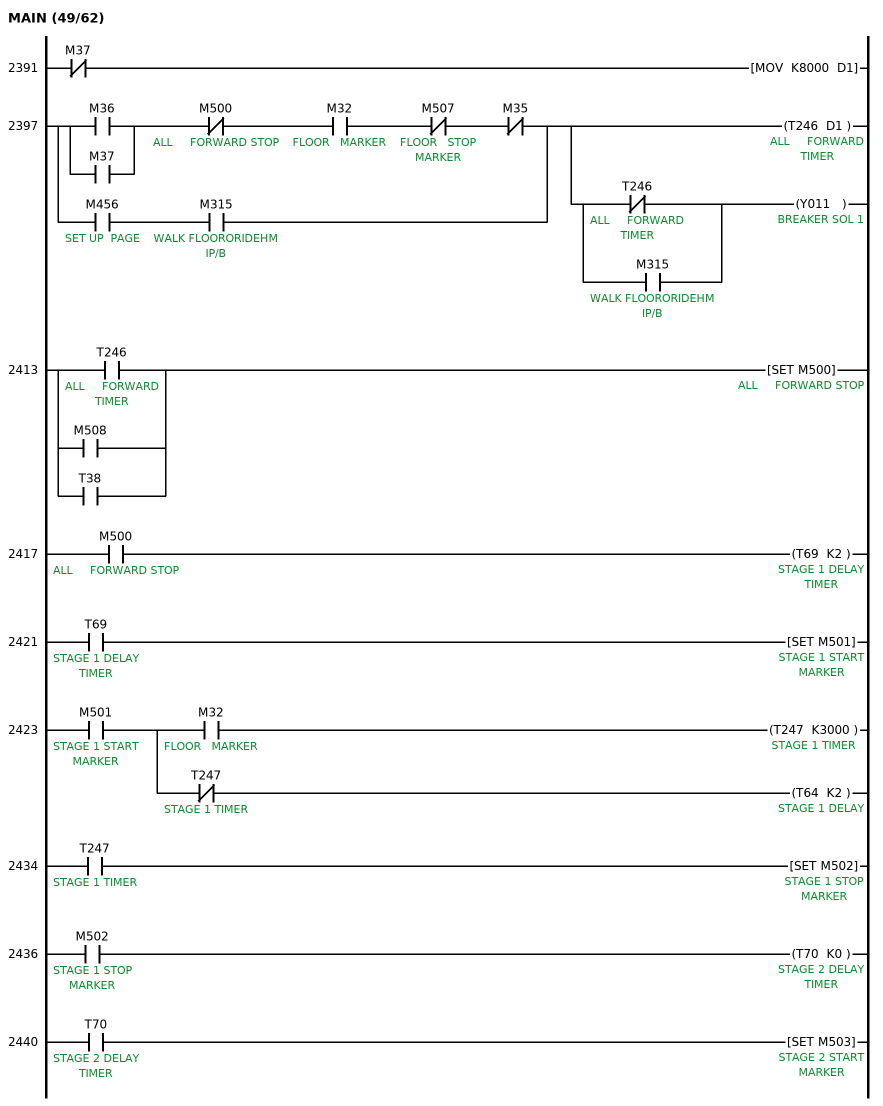
2391  LDI     M37
      MOV     K8000 D1
2397  LD      M36
      OR      M37
      ANI     M500  ; ALL     FORWARD STOP
      AND     M32  ; FLOOR   MARKER
      ANI     M507  ; FLOOR   STOP    MARKER
      ANI     M35
      LD      M456  ; SET UP  PAGE
      AND     M315  ; WALK FLOORORIDEHMIP/B
      ORB
      OUT     T246 D1  ; ALL     FORWARD TIMER
      LDI     T246  ; ALL     FORWARD TIMER
      OR      M315  ; WALK FLOORORIDEHMIP/B
      ANB
      OUT     Y011  ; BREAKER SOL 1
2413  LD      T246  ; ALL     FORWARD TIMER
      OR      M508
      OR      T38
      SET     M500  ; ALL     FORWARD STOP
2417  LD      M500  ; ALL     FORWARD STOP
      OUT     T69 K2  ; STAGE 1 DELAY   TIMER
2421  LD      T69  ; STAGE 1 DELAY   TIMER
      SET     M501  ; STAGE 1 START   MARKER
2423  LD      M501  ; STAGE 1 START   MARKER
      MPS
      AND     M32  ; FLOOR   MARKER
      OUT     T247 K3000  ; STAGE 1 TIMER
      MPP
      ANI     T247  ; STAGE 1 TIMER
      OUT     T64 K2  ; STAGE 1 DELAY
2434  LD      T247  ; STAGE 1 TIMER
      SET     M502  ; STAGE 1 STOP    MARKER
2436  LD      M502  ; STAGE 1 STOP    MARKER
      OUT     T70 K0  ; STAGE 2 DELAY   TIMER
2440  LD      T70  ; STAGE 2 DELAY   TIMER
      SET     M503  ; STAGE 2 START   MARKER
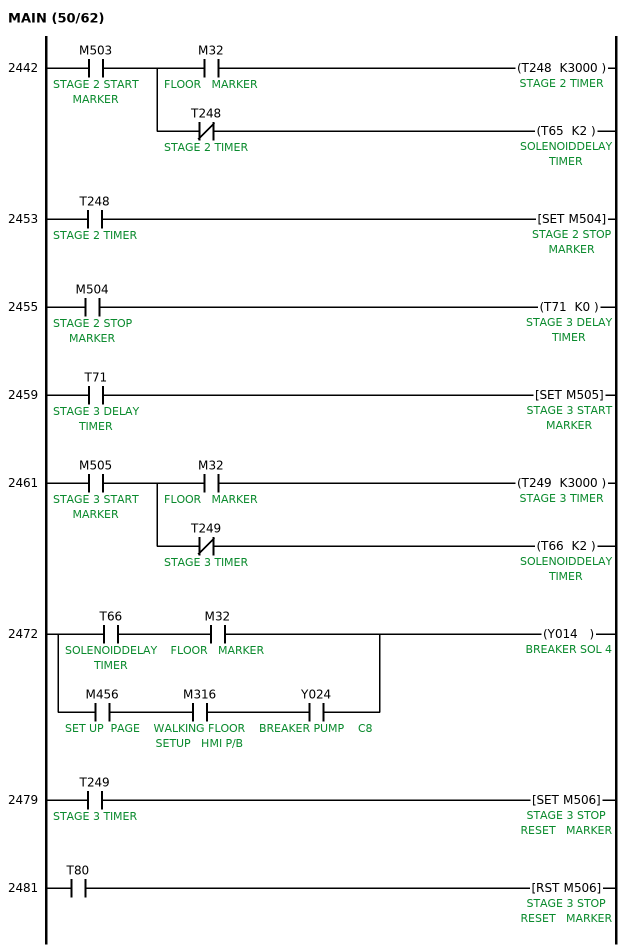
2442  LD      M503  ; STAGE 2 START   MARKER
      MPS
      AND     M32  ; FLOOR   MARKER
      OUT     T248 K3000  ; STAGE 2 TIMER
      MPP
      ANI     T248  ; STAGE 2 TIMER
      OUT     T65 K2  ; SOLENOIDDELAY   TIMER
2453  LD      T248  ; STAGE 2 TIMER
      SET     M504  ; STAGE 2 STOP    MARKER
2455  LD      M504  ; STAGE 2 STOP    MARKER
      OUT     T71 K0  ; STAGE 3 DELAY   TIMER
2459  LD      T71  ; STAGE 3 DELAY   TIMER
      SET     M505  ; STAGE 3 START   MARKER
2461  LD      M505  ; STAGE 3 START   MARKER
      MPS
      AND     M32  ; FLOOR   MARKER
      OUT     T249 K3000  ; STAGE 3 TIMER
      MPP
      ANI     T249  ; STAGE 3 TIMER
      OUT     T66 K2  ; SOLENOIDDELAY   TIMER
2472  LD      T66  ; SOLENOIDDELAY   TIMER
      AND     M32  ; FLOOR   MARKER
      LD      M456  ; SET UP  PAGE
      AND     M316  ; WALKING FLOOR   SETUP   HMI P/B
      AND     Y024  ; BREAKER PUMP    C8
      ORB
      OUT     Y014  ; BREAKER SOL 4
2479  LD      T249  ; STAGE 3 TIMER
      SET     M506  ; STAGE 3 STOP    RESET   MARKER
2481  LD      T80
      RST     M506  ; STAGE 3 STOP    RESET   MARKER
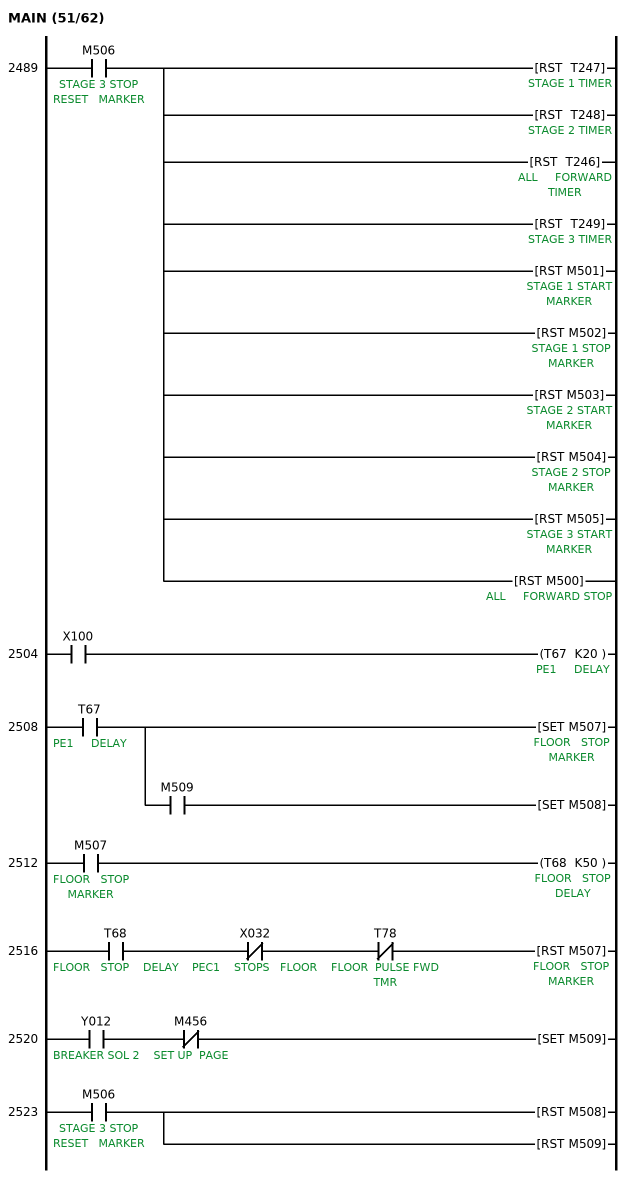
2489  LD      M506  ; STAGE 3 STOP    RESET   MARKER
      RST     T247  ; STAGE 1 TIMER
      RST     T248  ; STAGE 2 TIMER
      RST     T246  ; ALL     FORWARD TIMER
      RST     T249  ; STAGE 3 TIMER
      RST     M501  ; STAGE 1 START   MARKER
      RST     M502  ; STAGE 1 STOP    MARKER
      RST     M503  ; STAGE 2 START   MARKER
      RST     M504  ; STAGE 2 STOP    MARKER
      RST     M505  ; STAGE 3 START   MARKER
      RST     M500  ; ALL     FORWARD STOP
2504  LD      X100
      OUT     T67 K20  ; PE1     DELAY
2508  LD      T67  ; PE1     DELAY
      SET     M507  ; FLOOR   STOP    MARKER
      AND     M509
      SET     M508
2512  LD      M507  ; FLOOR   STOP    MARKER
      OUT     T68 K50  ; FLOOR   STOP    DELAY
2516  LD      T68  ; FLOOR   STOP    DELAY
      ANI     X032  ; PEC1    STOPS   FLOOR
      ANI     T78  ; FLOOR  PULSE FWD TMR
      RST     M507  ; FLOOR   STOP    MARKER
2520  LD      Y012  ; BREAKER SOL 2
      ANI     M456  ; SET UP  PAGE
      SET     M509
2523  LD      M506  ; STAGE 3 STOP    RESET   MARKER
      RST     M508
      RST     M509
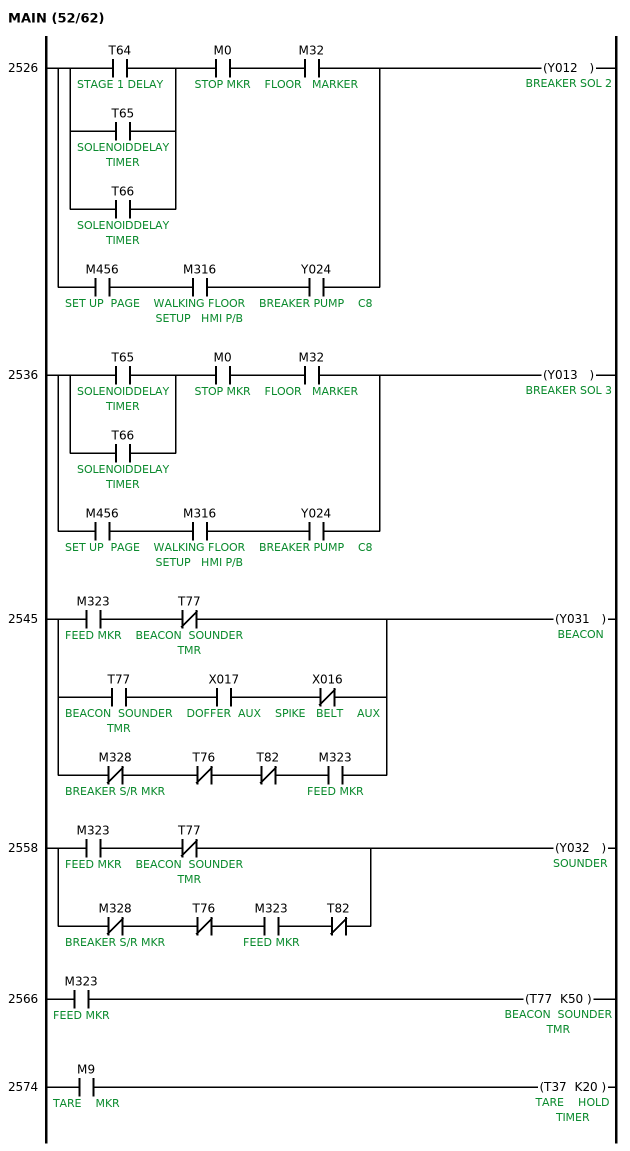
2526  LD      T64  ; STAGE 1 DELAY
      OR      T65  ; SOLENOIDDELAY   TIMER
      OR      T66  ; SOLENOIDDELAY   TIMER
      AND     M0  ; STOP MKR
      AND     M32  ; FLOOR   MARKER
      LD      M456  ; SET UP  PAGE
      AND     M316  ; WALKING FLOOR   SETUP   HMI P/B
      AND     Y024  ; BREAKER PUMP    C8
      ORB
      OUT     Y012  ; BREAKER SOL 2
2536  LD      T65  ; SOLENOIDDELAY   TIMER
      OR      T66  ; SOLENOIDDELAY   TIMER
      AND     M0  ; STOP MKR
      AND     M32  ; FLOOR   MARKER
      LD      M456  ; SET UP  PAGE
      AND     M316  ; WALKING FLOOR   SETUP   HMI P/B
      AND     Y024  ; BREAKER PUMP    C8
      ORB
      OUT     Y013  ; BREAKER SOL 3
2545  LD      M323  ; FEED MKR
      ANI     T77  ; BEACON  SOUNDER TMR
      LD      T77  ; BEACON  SOUNDER TMR
      AND     X017  ; DOFFER  AUX
      ANI     X016  ; SPIKE   BELT    AUX
      ORB
      LDI     M328  ; BREAKER S/R MKR
      ANI     T76
      ANI     T82
      AND     M323  ; FEED MKR
      ORB
      OUT     Y031  ; BEACON
2558  LD      M323  ; FEED MKR
      ANI     T77  ; BEACON  SOUNDER TMR
      LDI     M328  ; BREAKER S/R MKR
      ANI     T76
      AND     M323  ; FEED MKR
      ANI     T82
      ORB
      OUT     Y032  ; SOUNDER
2566  LD      M323  ; FEED MKR
      OUT     T77 K50  ; BEACON  SOUNDER TMR
2574  LD      M9  ; TARE    MKR
      OUT     T37 K20  ; TARE    HOLD    TIMER
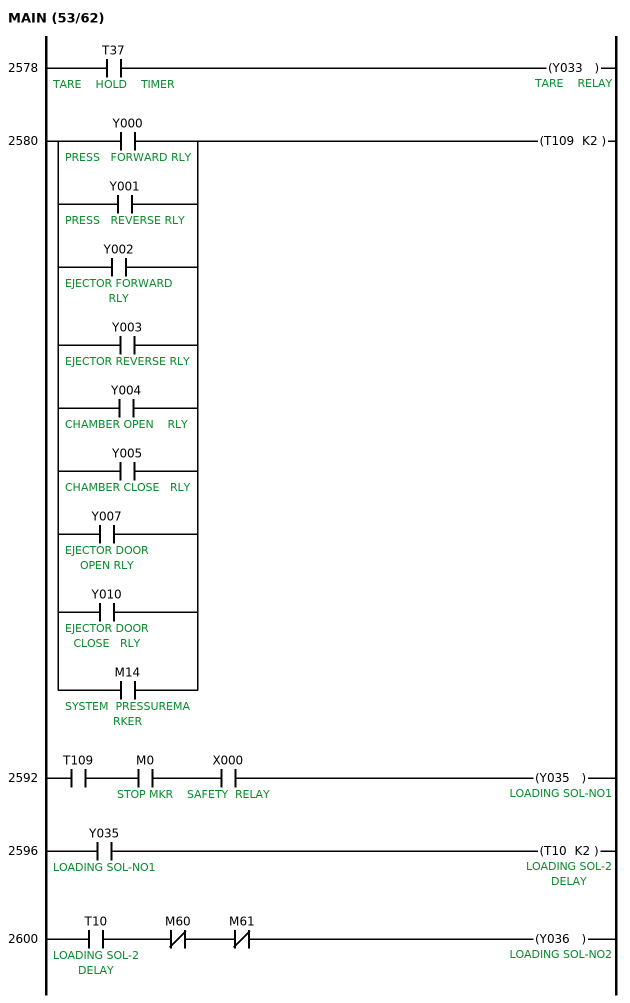
2578  LD      T37  ; TARE    HOLD    TIMER
      OUT     Y033  ; TARE    RELAY
2580  LD      Y000  ; PRESS   FORWARD RLY
      OR      Y001  ; PRESS   REVERSE RLY
      OR      Y002  ; EJECTOR FORWARD RLY
      OR      Y003  ; EJECTOR REVERSE RLY
      OR      Y004  ; CHAMBER OPEN    RLY
      OR      Y005  ; CHAMBER CLOSE   RLY
      OR      Y007  ; EJECTOR DOOR    OPEN RLY
      OR      Y010  ; EJECTOR DOOR    CLOSE   RLY
      OR      M14  ; SYSTEM  PRESSUREMARKER
      OUT     T109 K2
2592  LD      T109
      AND     M0  ; STOP MKR
      AND     X000  ; SAFETY  RELAY
      OUT     Y035  ; LOADING SOL-NO1
2596  LD      Y035  ; LOADING SOL-NO1
      OUT     T10 K2  ; LOADING SOL-2   DELAY
2600  LD      T10  ; LOADING SOL-2   DELAY
      ANI     M60
      ANI     M61
      OUT     Y036  ; LOADING SOL-NO2
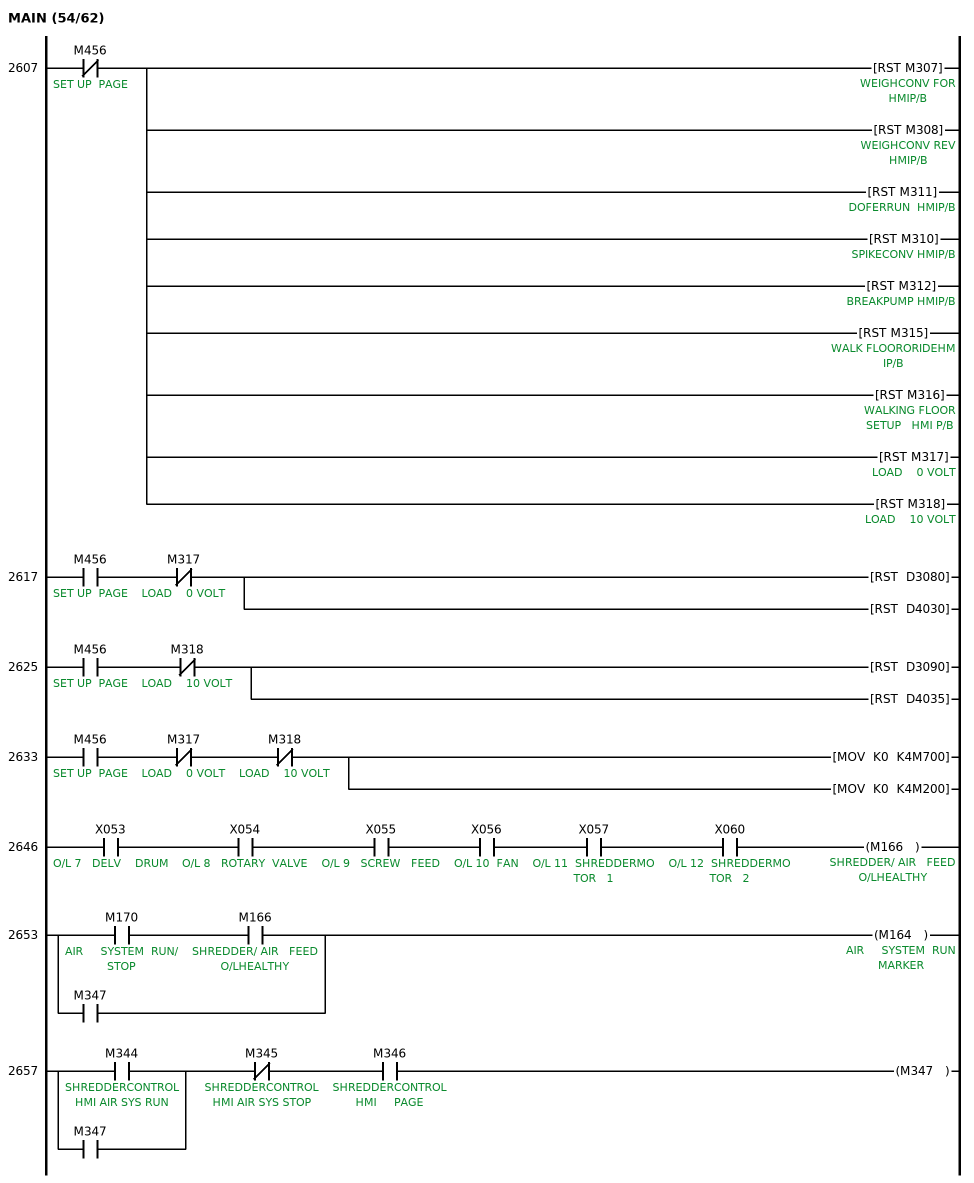
2607  LDI     M456  ; SET UP  PAGE
      RST     M307  ; WEIGHCONV FOR   HMIP/B
      RST     M308  ; WEIGHCONV REV   HMIP/B
      RST     M311  ; DOFERRUN  HMIP/B
      RST     M310  ; SPIKECONV HMIP/B
      RST     M312  ; BREAKPUMP HMIP/B
      RST     M315  ; WALK FLOORORIDEHMIP/B
      RST     M316  ; WALKING FLOOR   SETUP   HMI P/B
      RST     M317  ; LOAD    0 VOLT
      RST     M318  ; LOAD    10 VOLT
2617  LD      M456  ; SET UP  PAGE
      ANI     M317  ; LOAD    0 VOLT
      RST     D3080
      RST     D4030
2625  LD      M456  ; SET UP  PAGE
      ANI     M318  ; LOAD    10 VOLT
      RST     D3090
      RST     D4035
2633  LD      M456  ; SET UP  PAGE
      ANI     M317  ; LOAD    0 VOLT
      ANI     M318  ; LOAD    10 VOLT
      MOV     K0 K4M700
      MOV     K0 K4M200
2646  LD      X053  ; O/L 7   DELV    DRUM
      AND     X054  ; O/L 8   ROTARY  VALVE
      AND     X055  ; O/L 9   SCREW   FEED
      AND     X056  ; O/L 10  FAN
      AND     X057  ; O/L 11  SHREDDERMOTOR   1
      AND     X060  ; O/L 12  SHREDDERMOTOR   2
      OUT     M166  ; SHREDDER/ AIR   FEED O/LHEALTHY
2653  LD      M170  ; AIR     SYSTEM  RUN/    STOP
      AND     M166  ; SHREDDER/ AIR   FEED O/LHEALTHY
      OR      M347
      OUT     M164  ; AIR     SYSTEM  RUN     MARKER
2657  LD      M344  ; SHREDDERCONTROL HMI AIR SYS RUN
      OR      M347
      ANI     M345  ; SHREDDERCONTROL HMI AIR SYS STOP
      AND     M346  ; SHREDDERCONTROL HMI     PAGE
      OUT     M347
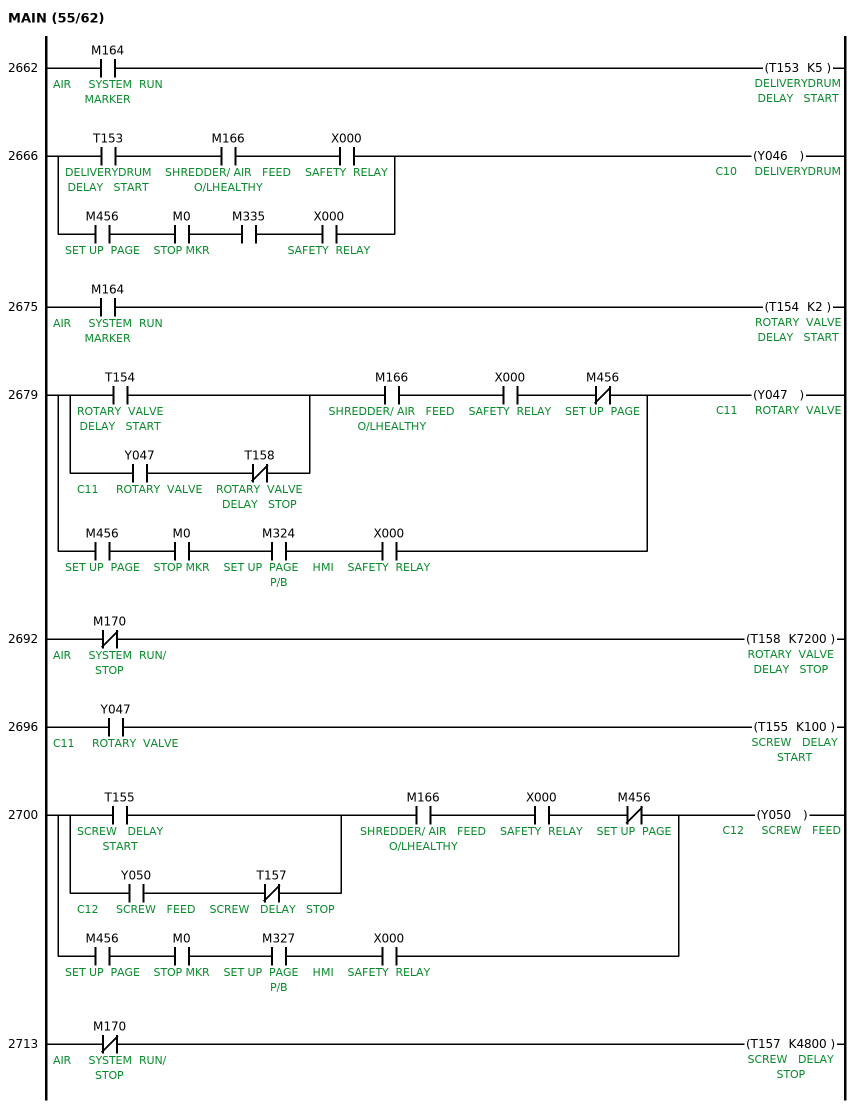
2662  LD      M164  ; AIR     SYSTEM  RUN     MARKER
      OUT     T153 K5  ; DELIVERYDRUM    DELAY   START
2666  LD      T153  ; DELIVERYDRUM    DELAY   START
      AND     M166  ; SHREDDER/ AIR   FEED O/LHEALTHY
      AND     X000  ; SAFETY  RELAY
      LD      M456  ; SET UP  PAGE
      AND     M0  ; STOP MKR
      AND     M335
      AND     X000  ; SAFETY  RELAY
      ORB
      OUT     Y046  ; C10     DELIVERYDRUM
2675  LD      M164  ; AIR     SYSTEM  RUN     MARKER
      OUT     T154 K2  ; ROTARY  VALVE   DELAY   START
2679  LD      T154  ; ROTARY  VALVE   DELAY   START
      LD      Y047  ; C11     ROTARY  VALVE
      ANI     T158  ; ROTARY  VALVE   DELAY   STOP
      ORB
      AND     M166  ; SHREDDER/ AIR   FEED O/LHEALTHY
      AND     X000  ; SAFETY  RELAY
      ANI     M456  ; SET UP  PAGE
      LD      M456  ; SET UP  PAGE
      AND     M0  ; STOP MKR
      AND     M324  ; SET UP  PAGE    HMI P/B
      AND     X000  ; SAFETY  RELAY
      ORB
      OUT     Y047  ; C11     ROTARY  VALVE
2692  LDI     M170  ; AIR     SYSTEM  RUN/    STOP
      OUT     T158 K7200  ; ROTARY  VALVE   DELAY   STOP
2696  LD      Y047  ; C11     ROTARY  VALVE
      OUT     T155 K100  ; SCREW   DELAY   START
2700  LD      T155  ; SCREW   DELAY   START
      LD      Y050  ; C12     SCREW   FEED
      ANI     T157  ; SCREW   DELAY   STOP
      ORB
      AND     M166  ; SHREDDER/ AIR   FEED O/LHEALTHY
      AND     X000  ; SAFETY  RELAY
      ANI     M456  ; SET UP  PAGE
      LD      M456  ; SET UP  PAGE
      AND     M0  ; STOP MKR
      AND     M327  ; SET UP  PAGE    HMI P/B
      AND     X000  ; SAFETY  RELAY
      ORB
      OUT     Y050  ; C12     SCREW   FEED
2713  LDI     M170  ; AIR     SYSTEM  RUN/    STOP
      OUT     T157 K4800  ; SCREW   DELAY   STOP
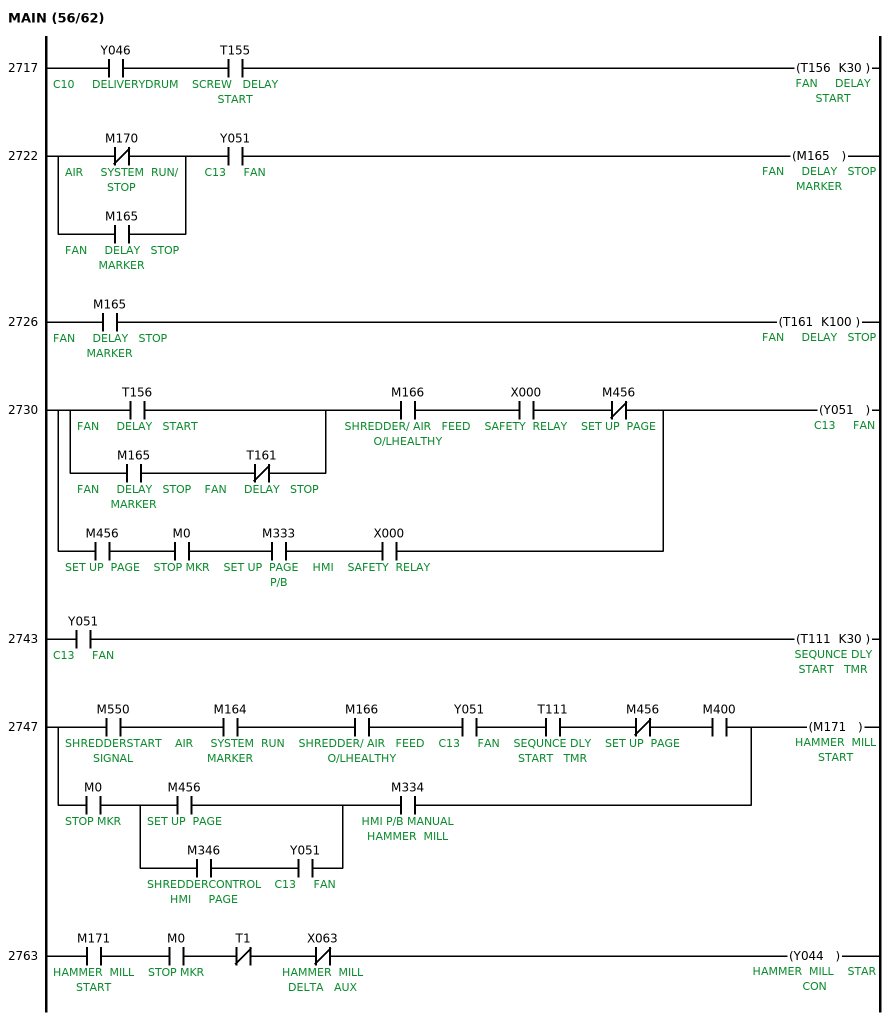
2717  LD      Y046  ; C10     DELIVERYDRUM
      AND     T155  ; SCREW   DELAY   START
      OUT     T156 K30  ; FAN     DELAY   START
2722  LDI     M170  ; AIR     SYSTEM  RUN/    STOP
      OR      M165  ; FAN     DELAY   STOP    MARKER
      AND     Y051  ; C13     FAN
      OUT     M165  ; FAN     DELAY   STOP    MARKER
2726  LD      M165  ; FAN     DELAY   STOP    MARKER
      OUT     T161 K100  ; FAN     DELAY   STOP
2730  LD      T156  ; FAN     DELAY   START
      LD      M165  ; FAN     DELAY   STOP    MARKER
      ANI     T161  ; FAN     DELAY   STOP
      ORB
      AND     M166  ; SHREDDER/ AIR   FEED O/LHEALTHY
      AND     X000  ; SAFETY  RELAY
      ANI     M456  ; SET UP  PAGE
      LD      M456  ; SET UP  PAGE
      AND     M0  ; STOP MKR
      AND     M333  ; SET UP  PAGE    HMI P/B
      AND     X000  ; SAFETY  RELAY
      ORB
      OUT     Y051  ; C13     FAN
2743  LD      Y051  ; C13     FAN
      OUT     T111 K30  ; SEQUNCE DLY     START   TMR
2747  LD      M550  ; SHREDDERSTART   SIGNAL
      AND     M164  ; AIR     SYSTEM  RUN     MARKER
      AND     M166  ; SHREDDER/ AIR   FEED O/LHEALTHY
      AND     Y051  ; C13     FAN
      AND     T111  ; SEQUNCE DLY     START   TMR
      ANI     M456  ; SET UP  PAGE
      AND     M400
      LD      M0  ; STOP MKR
      LD      M456  ; SET UP  PAGE
      LD      M346  ; SHREDDERCONTROL HMI     PAGE
      AND     Y051  ; C13     FAN
      ORB
      ANB
      AND     M334  ; HMI P/B MANUAL  HAMMER  MILL
      ORB
      OUT     M171  ; HAMMER  MILL    START
2763  LD      M171  ; HAMMER  MILL    START
      AND     M0  ; STOP MKR
      ANI     T1
      ANI     X063  ; HAMMER  MILL    DELTA   AUX
      OUT     Y044  ; HAMMER  MILL    STAR    CON
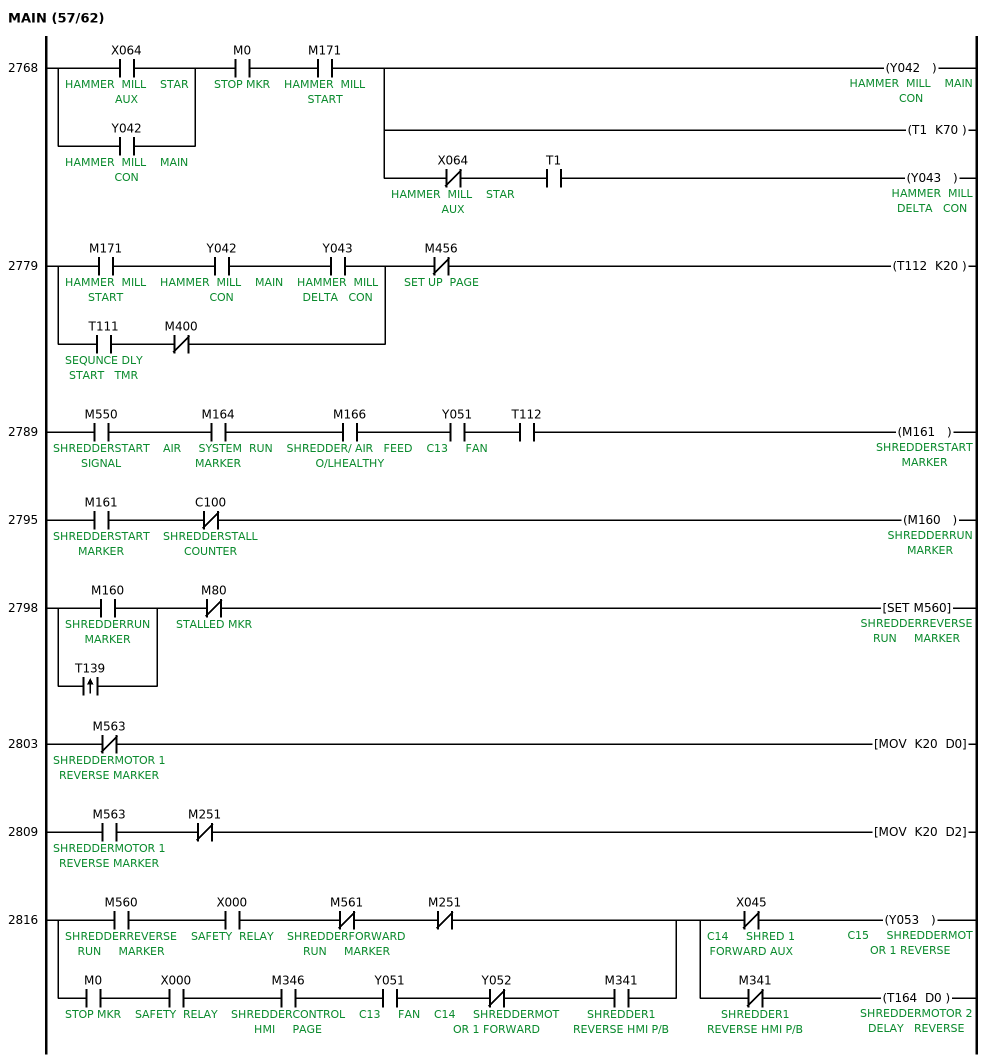
2768  LD      X064  ; HAMMER  MILL    STAR    AUX
      OR      Y042  ; HAMMER  MILL    MAIN    CON
      AND     M0  ; STOP MKR
      AND     M171  ; HAMMER  MILL    START
      OUT     Y042  ; HAMMER  MILL    MAIN    CON
      OUT     T1 K70
      ANI     X064  ; HAMMER  MILL    STAR    AUX
      AND     T1
      OUT     Y043  ; HAMMER  MILL    DELTA   CON
2779  LD      M171  ; HAMMER  MILL    START
      AND     Y042  ; HAMMER  MILL    MAIN    CON
      AND     Y043  ; HAMMER  MILL    DELTA   CON
      LD      T111  ; SEQUNCE DLY     START   TMR
      ANI     M400
      ORB
      ANI     M456  ; SET UP  PAGE
      OUT     T112 K20
2789  LD      M550  ; SHREDDERSTART   SIGNAL
      AND     M164  ; AIR     SYSTEM  RUN     MARKER
      AND     M166  ; SHREDDER/ AIR   FEED O/LHEALTHY
      AND     Y051  ; C13     FAN
      AND     T112
      OUT     M161  ; SHREDDERSTART   MARKER
2795  LD      M161  ; SHREDDERSTART   MARKER
      ANI     C100  ; SHREDDERSTALL   COUNTER
      OUT     M160  ; SHREDDERRUN     MARKER
2798  LD      M160  ; SHREDDERRUN     MARKER
      ORP     T139
      ANI     M80  ; STALLED MKR
      SET     M560  ; SHREDDERREVERSE RUN     MARKER
2803  LDI     M563  ; SHREDDERMOTOR 1 REVERSE MARKER
      MOV     K20 D0
2809  LD      M563  ; SHREDDERMOTOR 1 REVERSE MARKER
      ANI     M251
      MOV     K20 D2
2816  LD      M560  ; SHREDDERREVERSE RUN     MARKER
      AND     X000  ; SAFETY  RELAY
      ANI     M561  ; SHREDDERFORWARD RUN     MARKER
      ANI     M251
      LD      M0  ; STOP MKR
      AND     X000  ; SAFETY  RELAY
      AND     M346  ; SHREDDERCONTROL HMI     PAGE
      AND     Y051  ; C13     FAN
      ANI     Y052  ; C14     SHREDDERMOTOR 1 FORWARD
      AND     M341  ; SHREDDER1       REVERSE HMI P/B
      ORB
      MPS
      ANI     X045  ; C14     SHRED 1 FORWARD AUX
      OUT     Y053  ; C15     SHREDDERMOTOR 1 REVERSE
      MPP
      ANI     M341  ; SHREDDER1       REVERSE HMI P/B
      OUT     T164 D0  ; SHREDDERMOTOR 2 DELAY   REVERSE
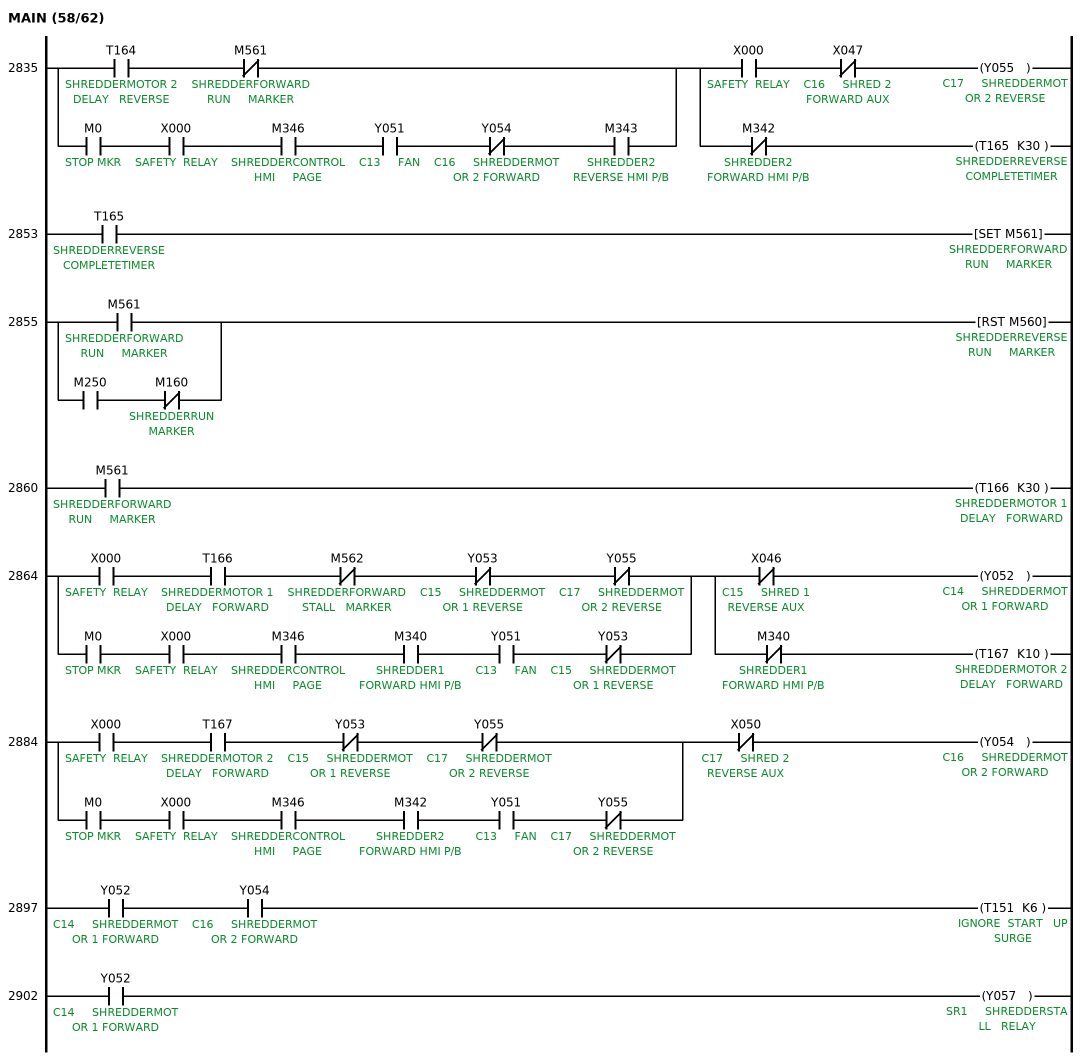
2835  LD      T164  ; SHREDDERMOTOR 2 DELAY   REVERSE
      ANI     M561  ; SHREDDERFORWARD RUN     MARKER
      LD      M0  ; STOP MKR
      AND     X000  ; SAFETY  RELAY
      AND     M346  ; SHREDDERCONTROL HMI     PAGE
      AND     Y051  ; C13     FAN
      ANI     Y054  ; C16     SHREDDERMOTOR 2 FORWARD
      AND     M343  ; SHREDDER2       REVERSE HMI P/B
      ORB
      MPS
      AND     X000  ; SAFETY  RELAY
      ANI     X047  ; C16     SHRED 2 FORWARD AUX
      OUT     Y055  ; C17     SHREDDERMOTOR 2 REVERSE
      MPP
      ANI     M342  ; SHREDDER2       FORWARD HMI P/B
      OUT     T165 K30  ; SHREDDERREVERSE COMPLETETIMER
2853  LD      T165  ; SHREDDERREVERSE COMPLETETIMER
      SET     M561  ; SHREDDERFORWARD RUN     MARKER
2855  LD      M561  ; SHREDDERFORWARD RUN     MARKER
      LD      M250
      ANI     M160  ; SHREDDERRUN     MARKER
      ORB
      RST     M560  ; SHREDDERREVERSE RUN     MARKER
2860  LD      M561  ; SHREDDERFORWARD RUN     MARKER
      OUT     T166 K30  ; SHREDDERMOTOR 1 DELAY   FORWARD
2864  LD      X000  ; SAFETY  RELAY
      AND     T166  ; SHREDDERMOTOR 1 DELAY   FORWARD
      ANI     M562  ; SHREDDERFORWARD STALL   MARKER
      ANI     Y053  ; C15     SHREDDERMOTOR 1 REVERSE
      ANI     Y055  ; C17     SHREDDERMOTOR 2 REVERSE
      LD      M0  ; STOP MKR
      AND     X000  ; SAFETY  RELAY
      AND     M346  ; SHREDDERCONTROL HMI     PAGE
      AND     M340  ; SHREDDER1       FORWARD HMI P/B
      AND     Y051  ; C13     FAN
      ANI     Y053  ; C15     SHREDDERMOTOR 1 REVERSE
      ORB
      MPS
      ANI     X046  ; C15     SHRED 1 REVERSE AUX
      OUT     Y052  ; C14     SHREDDERMOTOR 1 FORWARD
      MPP
      ANI     M340  ; SHREDDER1       FORWARD HMI P/B
      OUT     T167 K10  ; SHREDDERMOTOR 2 DELAY   FORWARD
2884  LD      X000  ; SAFETY  RELAY
      AND     T167  ; SHREDDERMOTOR 2 DELAY   FORWARD
      ANI     Y053  ; C15     SHREDDERMOTOR 1 REVERSE
      ANI     Y055  ; C17     SHREDDERMOTOR 2 REVERSE
      LD      M0  ; STOP MKR
      AND     X000  ; SAFETY  RELAY
      AND     M346  ; SHREDDERCONTROL HMI     PAGE
      AND     M342  ; SHREDDER2       FORWARD HMI P/B
      AND     Y051  ; C13     FAN
      ANI     Y055  ; C17     SHREDDERMOTOR 2 REVERSE
      ORB
      ANI     X050  ; C17     SHRED 2 REVERSE AUX
      OUT     Y054  ; C16     SHREDDERMOTOR 2 FORWARD
2897  LD      Y052  ; C14     SHREDDERMOTOR 1 FORWARD
      AND     Y054  ; C16     SHREDDERMOTOR 2 FORWARD
      OUT     T151 K6  ; IGNORE  START   UP      SURGE
2902  LD      Y052  ; C14     SHREDDERMOTOR 1 FORWARD
      OUT     Y057  ; SR1     SHREDDERSTALL   RELAY
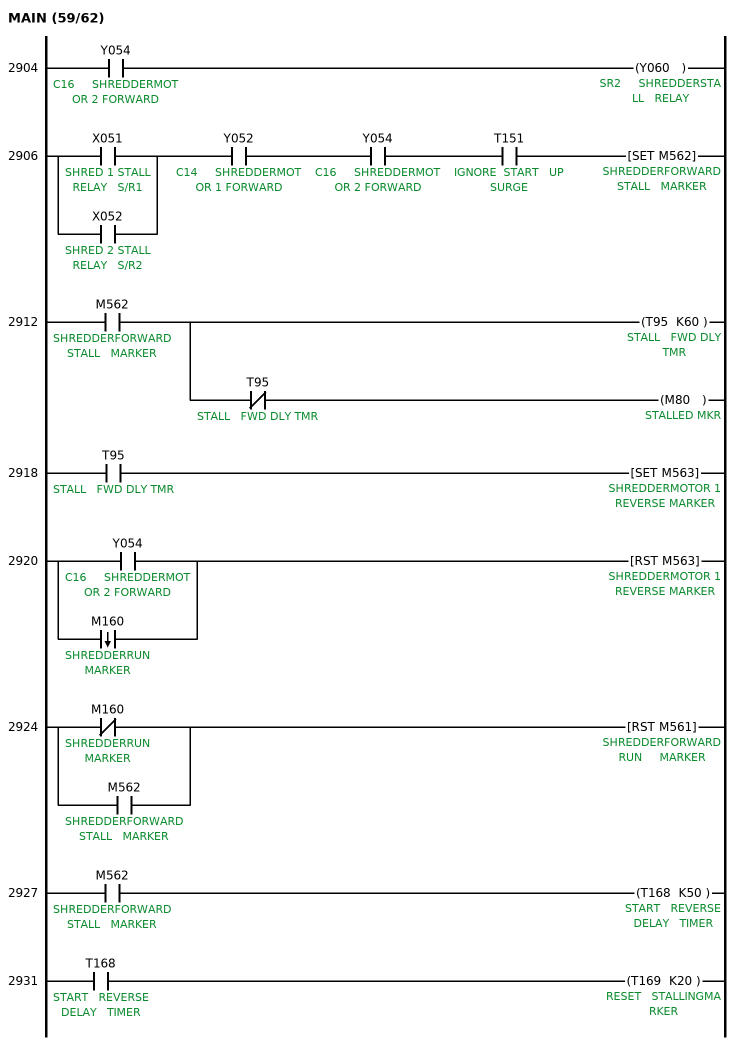
2904  LD      Y054  ; C16     SHREDDERMOTOR 2 FORWARD
      OUT     Y060  ; SR2     SHREDDERSTALL   RELAY
2906  LD      X051  ; SHRED 1 STALL   RELAY   S/R1
      OR      X052  ; SHRED 2 STALL   RELAY   S/R2
      AND     Y052  ; C14     SHREDDERMOTOR 1 FORWARD
      AND     Y054  ; C16     SHREDDERMOTOR 2 FORWARD
      AND     T151  ; IGNORE  START   UP      SURGE
      SET     M562  ; SHREDDERFORWARD STALL   MARKER
2912  LD      M562  ; SHREDDERFORWARD STALL   MARKER
      OUT     T95 K60  ; STALL   FWD DLY TMR
      ANI     T95  ; STALL   FWD DLY TMR
      OUT     M80  ; STALLED MKR
2918  LD      T95  ; STALL   FWD DLY TMR
      SET     M563  ; SHREDDERMOTOR 1 REVERSE MARKER
2920  LD      Y054  ; C16     SHREDDERMOTOR 2 FORWARD
      ORF     M160  ; SHREDDERRUN     MARKER
      RST     M563  ; SHREDDERMOTOR 1 REVERSE MARKER
2924  LDI     M160  ; SHREDDERRUN     MARKER
      OR      M562  ; SHREDDERFORWARD STALL   MARKER
      RST     M561  ; SHREDDERFORWARD RUN     MARKER
2927  LD      M562  ; SHREDDERFORWARD STALL   MARKER
      OUT     T168 K50  ; START   REVERSE DELAY   TIMER
2931  LD      T168  ; START   REVERSE DELAY   TIMER
      OUT     T169 K20  ; RESET   STALLINGMARKER
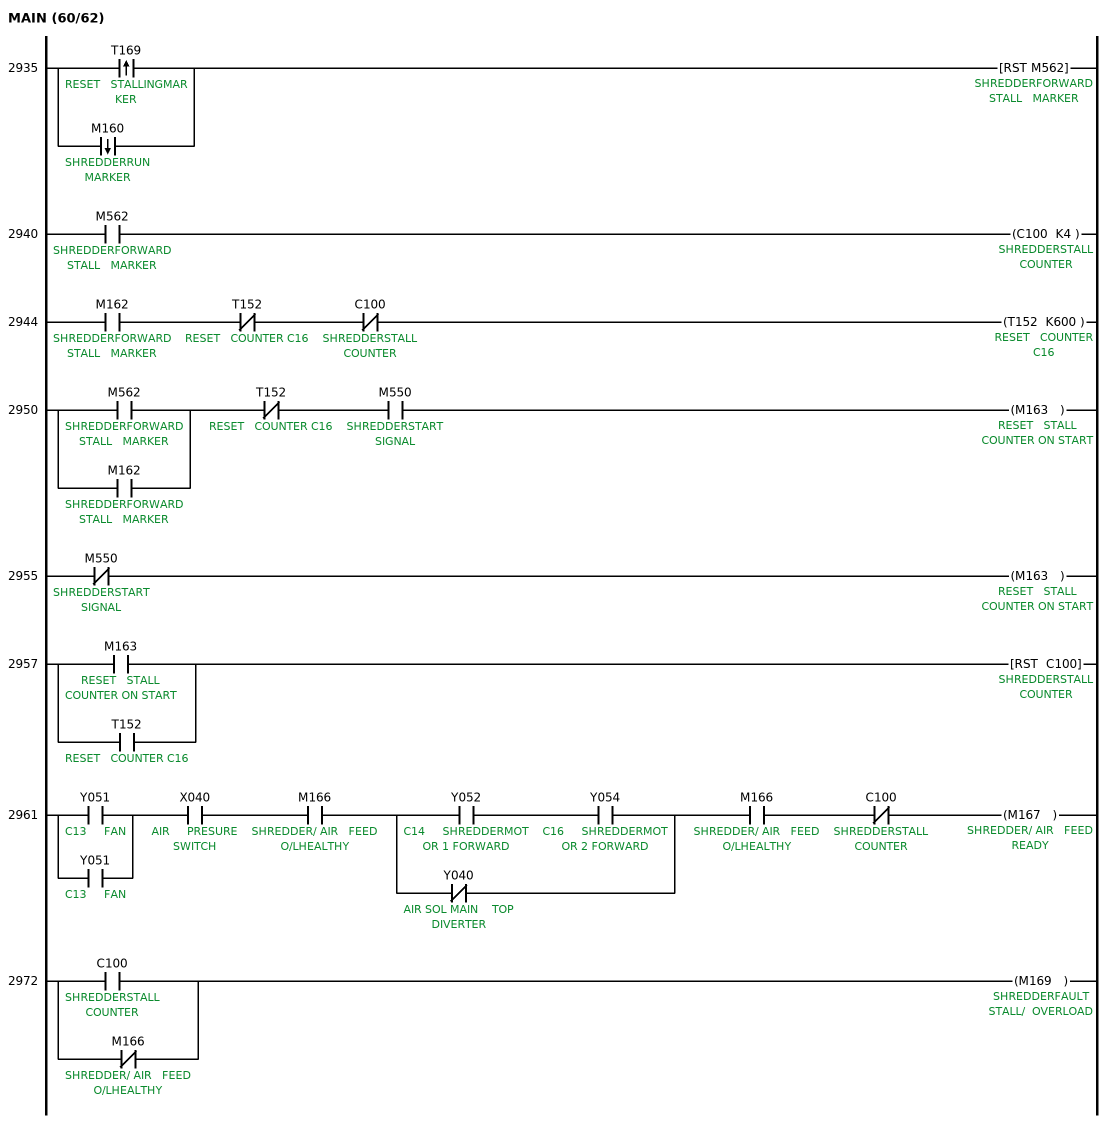
2935  LDP     T169  ; RESET   STALLINGMARKER
      ORF     M160  ; SHREDDERRUN     MARKER
      RST     M562  ; SHREDDERFORWARD STALL   MARKER
2940  LD      M562  ; SHREDDERFORWARD STALL   MARKER
      OUT     C100 K4  ; SHREDDERSTALL   COUNTER
2944  LD      M162  ; SHREDDERFORWARD STALL   MARKER
      ANI     T152  ; RESET   COUNTER C16
      ANI     C100  ; SHREDDERSTALL   COUNTER
      OUT     T152 K600  ; RESET   COUNTER C16
2950  LD      M562  ; SHREDDERFORWARD STALL   MARKER
      OR      M162  ; SHREDDERFORWARD STALL   MARKER
      ANI     T152  ; RESET   COUNTER C16
      AND     M550  ; SHREDDERSTART   SIGNAL
      OUT     M163  ; RESET   STALL   COUNTER ON START
2955  LDI     M550  ; SHREDDERSTART   SIGNAL
      OUT     M163  ; RESET   STALL   COUNTER ON START
2957  LD      M163  ; RESET   STALL   COUNTER ON START
      OR      T152  ; RESET   COUNTER C16
      RST     C100  ; SHREDDERSTALL   COUNTER
2961  LD      Y051  ; C13     FAN
      OR      Y051  ; C13     FAN
      AND     X040  ; AIR     PRESURE SWITCH
      AND     M166  ; SHREDDER/ AIR   FEED O/LHEALTHY
      LD      Y052  ; C14     SHREDDERMOTOR 1 FORWARD
      AND     Y054  ; C16     SHREDDERMOTOR 2 FORWARD
      ORI     Y040  ; AIR SOL MAIN    TOP     DIVERTER
      ANB
      AND     M166  ; SHREDDER/ AIR   FEED O/LHEALTHY
      ANI     C100  ; SHREDDERSTALL   COUNTER
      OUT     M167  ; SHREDDER/ AIR   FEED    READY
2972  LD      C100  ; SHREDDERSTALL   COUNTER
      ORI     M166  ; SHREDDER/ AIR   FEED O/LHEALTHY
      OUT     M169  ; SHREDDERFAULT   STALL/  OVERLOAD
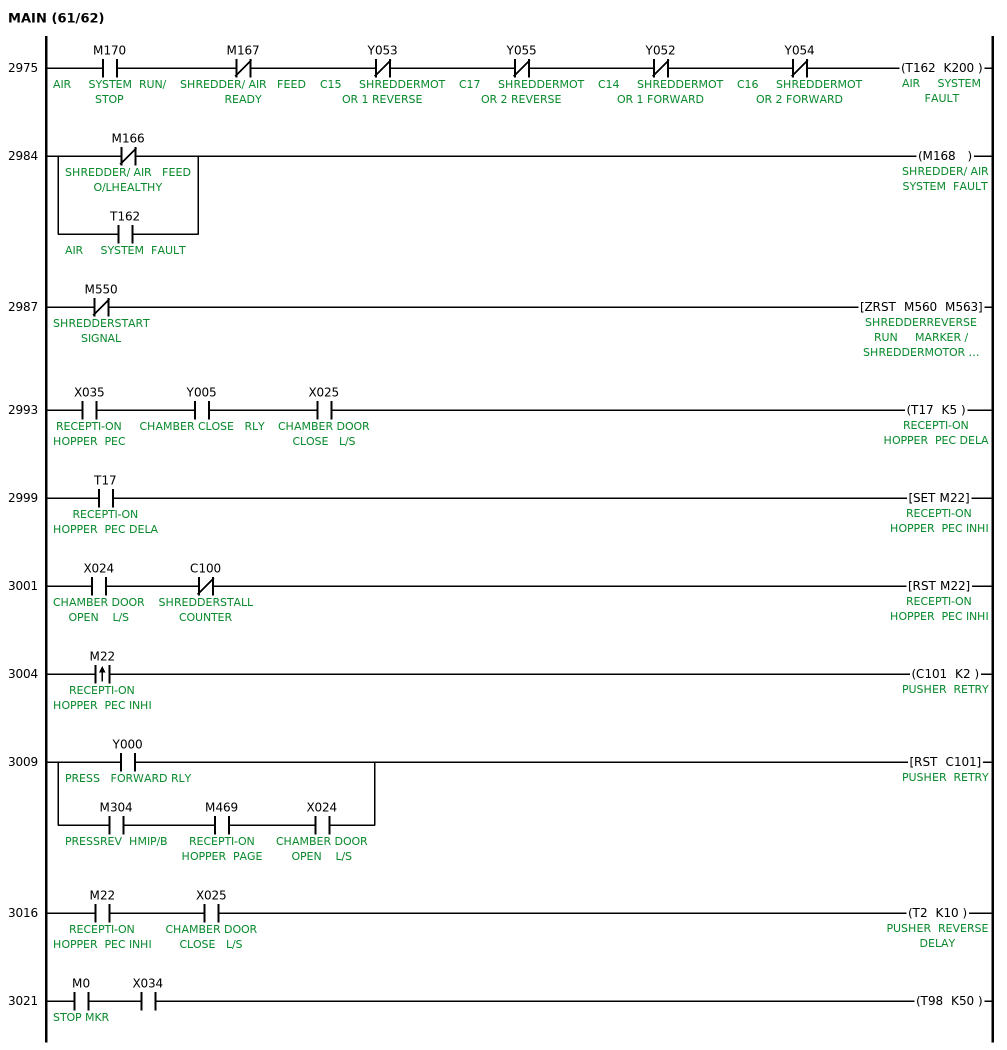
2975  LD      M170  ; AIR     SYSTEM  RUN/    STOP
      ANI     M167  ; SHREDDER/ AIR   FEED    READY
      ANI     Y053  ; C15     SHREDDERMOTOR 1 REVERSE
      ANI     Y055  ; C17     SHREDDERMOTOR 2 REVERSE
      ANI     Y052  ; C14     SHREDDERMOTOR 1 FORWARD
      ANI     Y054  ; C16     SHREDDERMOTOR 2 FORWARD
      OUT     T162 K200  ; AIR     SYSTEM  FAULT
2984  LDI     M166  ; SHREDDER/ AIR   FEED O/LHEALTHY
      OR      T162  ; AIR     SYSTEM  FAULT
      OUT     M168  ; SHREDDER/ AIR   SYSTEM  FAULT
2987  LDI     M550  ; SHREDDERSTART   SIGNAL
      ZRST    M560 M563
2993  LD      X035  ; RECEPTI-ON      HOPPER  PEC
      AND     Y005  ; CHAMBER CLOSE   RLY
      AND     X025  ; CHAMBER DOOR    CLOSE   L/S
      OUT     T17 K5  ; RECEPTI-ON      HOPPER  PEC DELA
2999  LD      T17  ; RECEPTI-ON      HOPPER  PEC DELA
      SET     M22  ; RECEPTI-ON      HOPPER  PEC INHI
3001  LD      X024  ; CHAMBER DOOR    OPEN    L/S
      ANI     C100  ; SHREDDERSTALL   COUNTER
      RST     M22  ; RECEPTI-ON      HOPPER  PEC INHI
3004  LDP     M22  ; RECEPTI-ON      HOPPER  PEC INHI
      OUT     C101 K2  ; PUSHER  RETRY
3009  LD      Y000  ; PRESS   FORWARD RLY
      LD      M304  ; PRESSREV  HMIP/B
      AND     M469  ; RECEPTI-ON      HOPPER  PAGE
      AND     X024  ; CHAMBER DOOR    OPEN    L/S
      ORB
      RST     C101  ; PUSHER  RETRY
3016  LD      M22  ; RECEPTI-ON      HOPPER  PEC INHI
      AND     X025  ; CHAMBER DOOR    CLOSE   L/S
      OUT     T2 K10  ; PUSHER  REVERSE DELAY
3021  LD      M0  ; STOP MKR
      AND     X034
      OUT     T98 K50
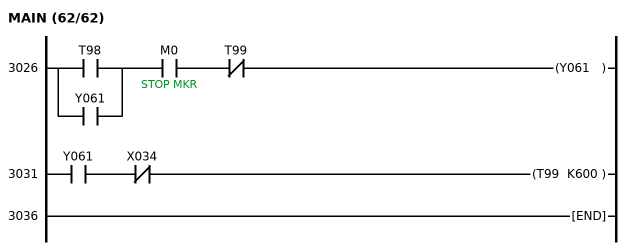
3026  LD      T98
      OR      Y061
      AND     M0  ; STOP MKR
      ANI     T99
      OUT     Y061
3031  LD      Y061
      ANI     X034
      OUT     T99 K600
3036  END
END_PROGRAM

// device comments not shown above
D1025  ; HMI  PSISET     POINT
M3  ; HOPPER
M172  ; SHREDDERSYSTEM  START/  STOP
M319  ; RESET   COUNTER
M424  ; EJECTOR RAM     REVERSE LIMIT
M425  ; EJECTOR DOOR    CLOSE   LIMIT
M426  ; PRESS   UP      LIMIT
M427  ; CHAMBER OPEN    LIMIT
M454  ; RECIPE  PAGE
M462  ; SYS PSI HMI MKR
X014  ; MAIN    CONTACT AUX     MCR1
X015  ; BREAKER PUMP    AUX
X026  ; CHAMBER DOOR    DOWN L/S
X041  ; C10     DELV    DRUM    AUX
X042  ; C11     ROTARY  VALVE   AUX
X043  ; C12     SCREW   FEED    AUX
X062  ; HAMMER  MILL    MAIN    AUX
X066  ; RECEPTI-ON      HOPPER  PEC
Y006  ; DE-COMP VALVE   RLY#
Y023  ; 24VDC   POWER   SUPPLY  C7
Y030  ; LOADING SOL
Y056  ; R23     RUN     SIGNAL
D102  ; HAMMER  MILL    AMPS
D128  ; CHAMBER DOOR    S-VALUE
D130  ; CHAMBER DOOR    FULL-SP
D132  ; CHAMBER DOOR    RAMP-DWN VALUE
D134  ; CHAMBER DOOR    RAMP-UP  RESULT
D136  ; CH-DOOR CLOSE   RAMP-DWN RESULT
D138  ; PRESS   DOWN    S-VALUE
D140  ; PRESS   DOWN    FULL-SP
D142  ; PRESS   DOWN    RAMP-DWN VALUE
D144  ; PRESS   DOWN    RAMP-UP RESULT
D146  ; PRESS   DOWN    RAMP-DWN RESULT
D148  ; EJECTOR DOOR    S-VALUE
D150  ; EJECTOR DOOR    FULL-SP
D152  ; EJECTOR DOOR    RAMP-DWN VALUE
D154  ; EJECTOR DOOR    RAMP-UP RESULT
D156  ; EJECTOR DOOR    RAMP-DWN RESULT
D158  ; EJECTOR RAM-FOR S-VALUE
D160  ; EJECTOR RAM-FOR FULL-SP
D162  ; EJECTOR RAM-FOR RAMP-DWN VALUE
D164  ; EJECTOR RAM-FOR RAMP-UP RESULT
D166  ; EJECTOR RAM-FOR RAMP-DWN RESULT
D168  ; EJECTOR RAM-REV S-VALUE
D170  ; EJECTOR RAM-REV FULL-SP
D172  ; EJECTOR RAM-REV RAMP-DWN VALUE
D174  ; EJECTOR RAM-REV RAMP-UP RESULT
D176  ; EJECTOR RAM-REV RAMP-DWN RESULT
D178  ; EJECTOR DOOR    S-VALUE
D180  ; EJECTOR DOOR    FULL-SP
D182  ; EJECTOR DOOR    RAMP-DWN VALUE
D184  ; EJECTOR DOOR    RAMP-UP RESULT
D186  ; EJECTOR DOOR    RAMP-DWN RESULT
D188  ; PRESS   UP    S-VALUE
D190  ; PRESS   UP    FULL-SP
D192  ; PRESS   UP    RAMP-DWN VALUE
D194  ; PRESS   UP    RAMP-UP RESULT
D196  ; PRESS   UP    RAMP-DWN RESULT
D198  ; CHAMBER DOOR    S-VALUE
D200  ; CHAMBER DOOR    FULL-SP
D202  ; CHAMBER DOOR    RAMP-DWN VALUE
D204  ; CHAMBER DOOR    RAMP-UP  RESULT
D206  ; CHAMBER DOOR   RAMP-DWN RESULT
D208  ; CHAMBER DOOR   RAMP-2   VALUE
D210  ; RAMP-2  RESULT  END
D212  ; PRESS   DOWN    PRESSURERAMP
D214  ; PRESS   DOWN    PRESSURERAMP RES
D216  ; EJECTOR FORWORD PRESSURERAMP
D218  ; EJECTOR FORWORD PRESSURERAMP RES
T160  ; SHREDDERDELAY   START
T250  ; SEQUENCECOMPLEAT
C205  ; RUN HOURHMI     DISPLAY
C234  ; bales produced resetable
C235  ; bales produced non-resetable
C240  ; HAY     BALE    TOTAL
